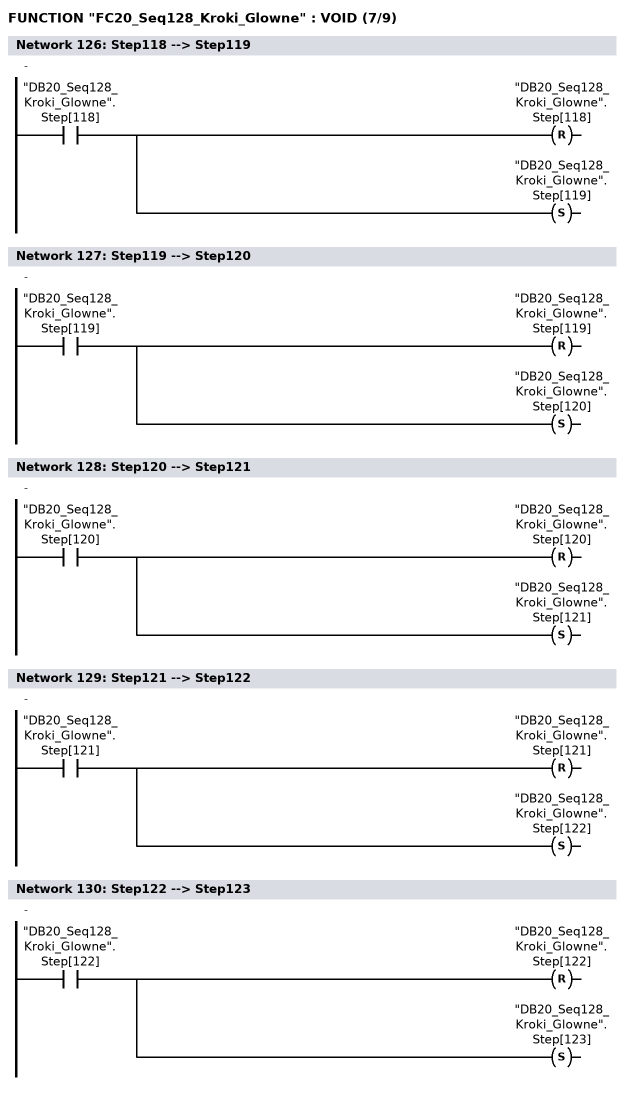
      A     "DB20_Seq128_Kroki_Glowne".Step[118];
      R     "DB20_Seq128_Kroki_Glowne".Step[118];
      S     "DB20_Seq128_Kroki_Glowne".Step[119];

NETWORK
TITLE = Step119 --> Step120
//-
      A     "DB20_Seq128_Kroki_Glowne".Step[119];
      R     "DB20_Seq128_Kroki_Glowne".Step[119];
      S     "DB20_Seq128_Kroki_Glowne".Step[120];

NETWORK
TITLE = Step120 --> Step121
//-
      A     "DB20_Seq128_Kroki_Glowne".Step[120];
      R     "DB20_Seq128_Kroki_Glowne".Step[120];
      S     "DB20_Seq128_Kroki_Glowne".Step[121];

NETWORK
TITLE = Step121 --> Step122
//-
      A     "DB20_Seq128_Kroki_Glowne".Step[121];
      R     "DB20_Seq128_Kroki_Glowne".Step[121];
      S     "DB20_Seq128_Kroki_Glowne".Step[122];

NETWORK
TITLE = Step122 --> Step123
//-
      A     "DB20_Seq128_Kroki_Glowne".Step[122];
      R     "DB20_Seq128_Kroki_Glowne".Step[122];
      S     "DB20_Seq128_Kroki_Glowne".Step[123];

NETWORK
TITLE = Step123 --> Step124
//-
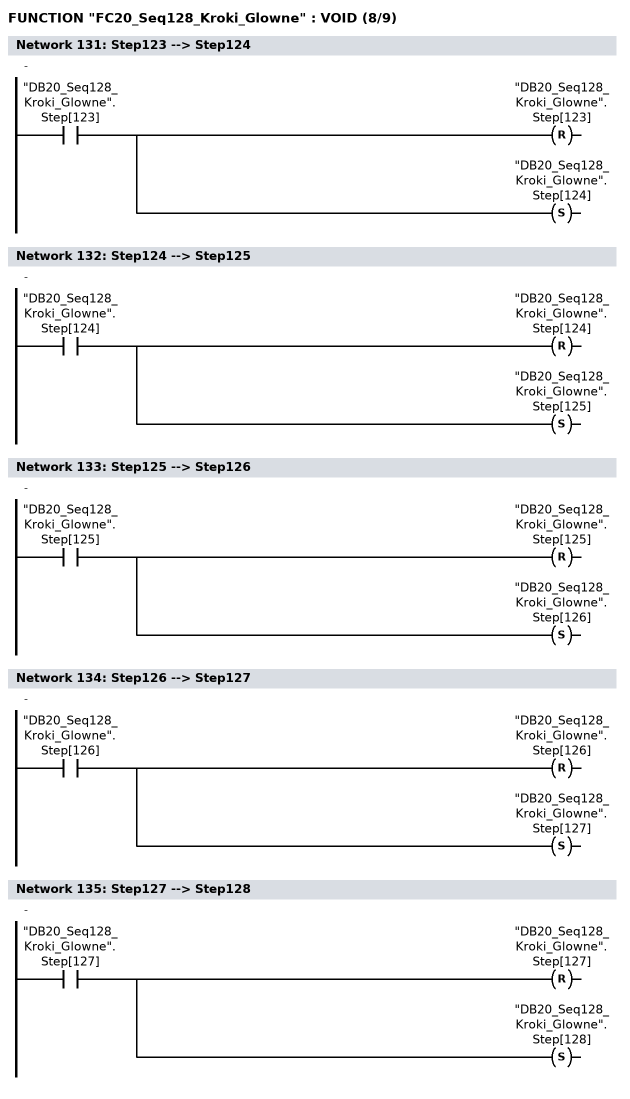
      A     "DB20_Seq128_Kroki_Glowne".Step[123];
      R     "DB20_Seq128_Kroki_Glowne".Step[123];
      S     "DB20_Seq128_Kroki_Glowne".Step[124];

NETWORK
TITLE = Step124 --> Step125
//-
      A     "DB20_Seq128_Kroki_Glowne".Step[124];
      R     "DB20_Seq128_Kroki_Glowne".Step[124];
      S     "DB20_Seq128_Kroki_Glowne".Step[125];

NETWORK
TITLE = Step125 --> Step126
//-
      A     "DB20_Seq128_Kroki_Glowne".Step[125];
      R     "DB20_Seq128_Kroki_Glowne".Step[125];
      S     "DB20_Seq128_Kroki_Glowne".Step[126];

NETWORK
TITLE = Step126 --> Step127
//-
      A     "DB20_Seq128_Kroki_Glowne".Step[126];
      R     "DB20_Seq128_Kroki_Glowne".Step[126];
      S     "DB20_Seq128_Kroki_Glowne".Step[127];

NETWORK
TITLE = Step127 --> Step128
//-
      A     "DB20_Seq128_Kroki_Glowne".Step[127];
      R     "DB20_Seq128_Kroki_Glowne".Step[127];
      S     "DB20_Seq128_Kroki_Glowne".Step[128];
NETWORK
TITLE =ZAPĘTLENIE
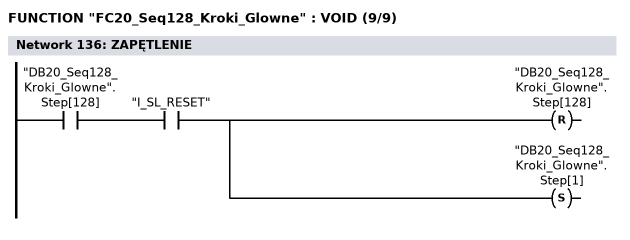

      A     "DB20_Seq128_Kroki_Glowne".Step[128];
      A     "I_SL_RESET";
      R     "DB20_Seq128_Kroki_Glowne".Step[128];
      S     "DB20_Seq128_Kroki_Glowne".Step[1];

END_FUNCTION

